(* PLC project descent, Dassault Systèmes ControlBuild 2024x *)
(* stored: creationDateTime 2023-10-03T11:13:44-01:00 *)

FUNCTION_BLOCK drill.descent
  VAR_INPUT
    acknowledgePB : BOOL := false;
  END_VAR
  VAR_INPUT
    slowAscent : BOOL := false;
    fastAscent : BOOL := false;
    slowDescent : BOOL := false;
    fastDescent : BOOL := false;
  END_VAR
  VAR_INPUT
    equipmentFault : BOOL := false;
  END_VAR
  VAR_OUTPUT
    motorFault : DINT := 0;
  END_VAR
  VAR_OUTPUT
    forward : BOOL := false;
    backward : BOOL := false;
    highSpeed : BOOL := false;
    lowSpeed : BOOL := false;
  END_VAR

INITIAL_STEP 10:
  COMPUTE_FUNCTION_BLOCKS(S);
END_STEP
TRANSITION FROM 10 TO 11
  := fastAscent AND (motorFault = 0);
END_TRANSITION
INITIAL_STEP 20:
END_STEP
TRANSITION FROM 20 TO 21
  := fastDescent AND (motorFault = 0);
END_TRANSITION
INITIAL_STEP 30:
END_STEP
TRANSITION FROM 30 TO 31
  := slowAscent AND (motorFault = 0);
END_TRANSITION
INITIAL_STEP 40:
END_STEP
TRANSITION FROM 40 TO 41
  := slowDescent AND (motorFault = 0);
END_TRANSITION
STEP 11:
  11_INLINE1(N);
END_STEP
ACTION 11_INLINE1:
  backward;
  highSpeed;
END_ACTION
TRANSITION FROM 11 TO 10
  := NOT fastAscent OR (motorFault > 0);
END_TRANSITION
STEP 21:
  21_INLINE2(N);
END_STEP
ACTION 21_INLINE2:
  forward;
  highSpeed;
END_ACTION
TRANSITION FROM 21 TO 20
  := NOT fastDescent OR (motorFault > 0);
END_TRANSITION
STEP 31:
  31_INLINE3(N);
END_STEP
ACTION 31_INLINE3:
  backward;
  lowSpeed;
END_ACTION
TRANSITION FROM 31 TO 30
  := NOT slowAscent OR (motorFault > 0);
END_TRANSITION
STEP 41:
  41_INLINE4(N);
END_STEP
ACTION 41_INLINE4:
  forward;
  lowSpeed;
END_ACTION
TRANSITION FROM 41 TO 40
  := NOT slowDescent OR (motorFault > 0);
END_TRANSITION
ACTION COMPUTE_FUNCTION_BLOCKS:  (* blocks drawn on the SFC sheet *)
  G1:
  G2:
  G3:
  G4:
END_ACTION

ACTION PreSFC:
IF((RE acknowledgePB)) THEN
	motorFault := 0;
END_IF;
IF((X21 OR X41) AND equipmentFault) THEN
	motorFault := 1;
END_IF;
IF((X31 OR X11) AND equipmentFault) THEN
	motorFault := 2;
END_IF;
IF ((X21 OR X11) AND equipmentFault) THEN
	motorFault := 3;
END_IF;
IF ((X41 OR X31) AND equipmentFault) THEN
	motorFault := 4;
END_IF;
END_ACTION
END_FUNCTION_BLOCK
